FUNCTION_BLOCK FB_FilterCombinations
VAR
    aThicknesses : ARRAY[1..nMAXIMUM_NUMBER_OF_THICKNESSES] OF LREAL;
    nFilterPositions : ARRAY[1..nMAXIMUM_NUMBER_OF_THICKNESSES] OF ARRAY[1..5] OF INT;
    nNumberOfThicknesses : UDINT;
END_VAR
VAR CONSTANT
    nMAXIMUM_NUMBER_OF_THICKNESSES : UDINT := 10000;
END_VAR


METHOD PUBLIC AddFilterCombination
VAR_INPUT
    fThickness : LREAL;
    aCombination : ARRAY[1..5] OF INT;
END_VAR

IF nNumberOfThicknesses >= nMAXIMUM_NUMBER_OF_THICKNESSES THEN
    RETURN;
END_IF

nNumberOfThicknesses := nNumberOfThicknesses + 1;
aThicknesses[nNumberOfThicknesses] := fThickness;
nFilterPositions[nNumberOfThicknesses] := aCombination;
END_METHOD


METHOD PUBLIC Reset

nNumberOfThicknesses := 0;

MEMSET(destAddr := ADR(aThicknesses),
       fillByte := 16#0,
       n := SIZEOF(aThicknesses));

MEMSET(destAddr := ADR(nFilterPositions),
       fillByte := 16#0,
       n := SIZEOF(nFilterPositions));
END_METHOD

END_FUNCTION_BLOCK

(* stored: Version 1.1.0.1
   POU FB_FilterCombinations: Id {4b240f92-978e-4d19-be0a-9ddef7b6361c}, SpecialFunc None
   Method AddFilterCombination: Id {f4eb5908-4a36-48dd-84ff-a98c52084b57}
   Method Reset: Id {912b6c75-b835-4fa2-8b93-0deeceaaf550} *)
